FUNCTION_BLOCK ClampInsertion
VAR_INPUT
	enable : BOOL;
END_VAR
VAR_OUTPUT
	slider : ServoECAT;
	screw : TeknicEIP;
	
	status : BOOL;
	contact : BOOL;
	
	home : BOOL;
	busy : BOOL;
	error : BOOL;
END_VAR
(*
this FB encapsulates a ServoECAT and TeknicEIP into a 2D insertion machine
normal operation should only use this FB's methods, but attributes and methods of the 2 components remain visible
*)

slider(
	bEnable:= enable, 
	home=> , 
	outerLimit=> , 
	innerLimit=> , 
	ready=> , 
	busy=> , 
	error=> , 
	homeSet=> );
	
screw(
	bEnable:= enable, 
	home=> , 
	outerLimit=> , 
	innerLimit=> , 
	done=> , 
	contact=> contact, 
	homeSet=> );

home := screw.home AND slider.home;
busy := slider.busy OR screw.busy;
error := slider.error OR screw.error;

METHOD alignTarget : BOOL
VAR_INPUT
	targetPos : REAL;
END_VAR
alignTarget := slider.moveAbsolute(position:= targetPos, fault=> );
END_METHOD

METHOD homingSequence : BOOL
IF NOT slider.homeSet THEN
	slider.homingSequence();
END_IF

IF NOT screw.homeSet THEN
	screw.homingSequence();
END_IF

homingSequence := slider.homeSet AND screw.homeSet;
END_METHOD

METHOD press : BOOL
VAR_INPUT
	//direction : BOOL; //direction (F = inwards, T = outwards)
	//distance : DINT;
END_VAR
screw.traverse(direction := FALSE);
END_METHOD

METHOD release : BOOL
VAR_INPUT
END_VAR
release := screw.traverse(direction := TRUE);
END_METHOD

METHOD slideContinuous : BOOL
VAR_INPUT
	direction : BOOL; //direction (F = inwards, T = outwards)
END_VAR
slideContinuous := slider.moveContinuous(direction);
END_METHOD

END_FUNCTION_BLOCK

(* stored: Version 1.1.0.1, ProductVersion 3.1.4024.11
   POU ClampInsertion: Id {a8054870-0722-4545-9a54-faef9caca0df}, SpecialFunc None
   Method alignTarget: Id {146b27b0-2ea0-4a44-8090-94a98937b16a}
   Method homingSequence: Id {3e0fa2d6-3807-446a-a1fe-017650352eb9}
   Method press: Id {e707c16a-c2a4-4550-814a-d7a5dbb9ebbc}
   Method release: Id {b125690b-923b-41e3-80da-f27e24ac2b0c}
   Method slideContinuous: Id {e1c7bb96-fb1a-45e9-b9a9-3ad3d62f4ef8} *)
